FUNCTION_BLOCK FB_2001_doublecookie
VAR_INPUT
	execute: BOOL;
END_VAR
VAR
	TIMERDONE: BOOL;
END_VAR

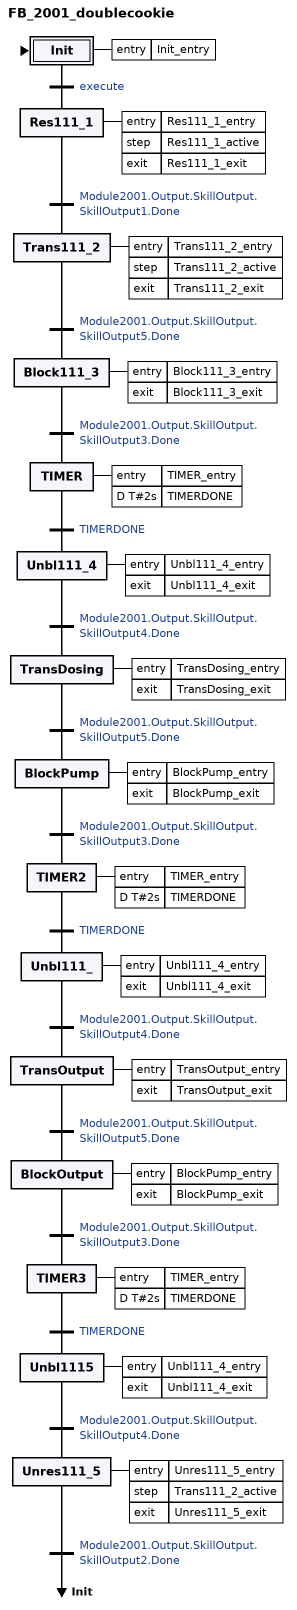
INITIAL_STEP Init:
    Init_entry(P1);  // entry action
END_STEP
TRANSITION FROM Init TO Res111_1
    := execute;
END_TRANSITION
STEP Res111_1:
    Res111_1_entry(P1);  // entry action
    Res111_1_active(N);  // step action
    Res111_1_exit(P0);  // exit action
END_STEP
TRANSITION FROM Res111_1 TO Trans111_2
    := Module2001.Output.SkillOutput.SkillOutput1.Done;
END_TRANSITION
STEP Trans111_2:
    Trans111_2_entry(P1);  // entry action
    Trans111_2_active(N);  // step action
    Trans111_2_exit(P0);  // exit action
END_STEP
TRANSITION FROM Trans111_2 TO Block111_3
    := Module2001.Output.SkillOutput.SkillOutput5.Done;
END_TRANSITION
STEP Block111_3:
    Block111_3_entry(P1);  // entry action
    Block111_3_exit(P0);  // exit action
END_STEP
TRANSITION FROM Block111_3 TO TIMER
    := Module2001.Output.SkillOutput.SkillOutput3.Done;
END_TRANSITION
STEP TIMER:
    TIMER_entry(P1);  // entry action
    TIMERDONE(D, T#2s);
END_STEP
TRANSITION FROM TIMER TO Unbl111_4
    := TIMERDONE;
END_TRANSITION
STEP Unbl111_4:
    Unbl111_4_entry(P1);  // entry action
    Unbl111_4_exit(P0);  // exit action
END_STEP
TRANSITION FROM Unbl111_4 TO TransDosing
    := Module2001.Output.SkillOutput.SkillOutput4.Done;
END_TRANSITION
STEP TransDosing:
    TransDosing_entry(P1);  // entry action
    TransDosing_exit(P0);  // exit action
END_STEP
TRANSITION FROM TransDosing TO BlockPump
    := Module2001.Output.SkillOutput.SkillOutput5.Done;
END_TRANSITION
STEP BlockPump:
    BlockPump_entry(P1);  // entry action
    BlockPump_exit(P0);  // exit action
END_STEP
TRANSITION FROM BlockPump TO TIMER2
    := Module2001.Output.SkillOutput.SkillOutput3.Done;
END_TRANSITION
STEP TIMER2:
    TIMER_entry(P1);  // entry action
    TIMERDONE(D, T#2s);
END_STEP
TRANSITION FROM TIMER2 TO Unbl111_
    := TIMERDONE;
END_TRANSITION
STEP Unbl111_:
    Unbl111_4_entry(P1);  // entry action
    Unbl111_4_exit(P0);  // exit action
END_STEP
TRANSITION FROM Unbl111_ TO TransOutput
    := Module2001.Output.SkillOutput.SkillOutput4.Done;
END_TRANSITION
STEP TransOutput:
    TransOutput_entry(P1);  // entry action
    TransOutput_exit(P0);  // exit action
END_STEP
TRANSITION FROM TransOutput TO BlockOutput
    := Module2001.Output.SkillOutput.SkillOutput5.Done;
END_TRANSITION
STEP BlockOutput:
    BlockPump_entry(P1);  // entry action
    BlockPump_exit(P0);  // exit action
END_STEP
TRANSITION FROM BlockOutput TO TIMER3
    := Module2001.Output.SkillOutput.SkillOutput3.Done;
END_TRANSITION
STEP TIMER3:
    TIMER_entry(P1);  // entry action
    TIMERDONE(D, T#2s);
END_STEP
TRANSITION FROM TIMER3 TO Unbl1115
    := TIMERDONE;
END_TRANSITION
STEP Unbl1115:
    Unbl111_4_entry(P1);  // entry action
    Unbl111_4_exit(P0);  // exit action
END_STEP
TRANSITION FROM Unbl1115 TO Unres111_5
    := Module2001.Output.SkillOutput.SkillOutput4.Done;
END_TRANSITION
STEP Unres111_5:
    Unres111_5_entry(P1);  // entry action
    Trans111_2_active(N);  // step action
    Unres111_5_exit(P0);  // exit action
END_STEP
TRANSITION FROM Unres111_5 TO Init
    := Module2001.Output.SkillOutput.SkillOutput2.Done;
END_TRANSITION

ACTION Block111_3_exit:
//BLOCKIEREN

Module2001.Input.SkillInput.SkillInput3.Execute := FALSE;
Module2001.Input.SkillInput.SkillInput3.ParameterInput.Parameterinput1.Value := 0; //TaskID
END_ACTION

ACTION TransDosing_entry:
//TRANSPORTIEREN

Module2001.Input.SkillInput.SkillInput5.Execute := TRUE;
Module2001.Input.SkillInput.SkillInput5.ParameterInput.Parameterinput1.Value := 3000; //X-Position
Module2001.Input.SkillInput.SkillInput5.ParameterInput.Parameterinput2.Value := 100;//90; //Z-Position
Module2001.Input.SkillInput.SkillInput5.ParameterInput.Parameterinput3.Value := 300; //Velocity
Module2001.Input.SkillInput.SkillInput5.ParameterInput.Parameterinput4.Value := 0; //Acceleration
END_ACTION

ACTION TransOutput_entry:
//TRANSPORTIEREN

Module2001.Input.SkillInput.SkillInput5.Execute := TRUE;
Module2001.Input.SkillInput.SkillInput5.ParameterInput.Parameterinput1.Value := 3300; //X-Position
Module2001.Input.SkillInput.SkillInput5.ParameterInput.Parameterinput2.Value := 110;//90; //Z-Position
Module2001.Input.SkillInput.SkillInput5.ParameterInput.Parameterinput3.Value := 300; //Velocity
Module2001.Input.SkillInput.SkillInput5.ParameterInput.Parameterinput4.Value := 0; //Acceleration
END_ACTION

ACTION TransOutput_exit:

Module2001.Input.SkillInput.SkillInput5.Execute := FALSE;
Module2001.Input.SkillInput.SkillInput5.ParameterInput.Parameterinput1.Value := 0; //X-Position
Module2001.Input.SkillInput.SkillInput5.ParameterInput.Parameterinput2.Value := 0; //Z-Position
Module2001.Input.SkillInput.SkillInput5.ParameterInput.Parameterinput3.Value := 0; //Velocity
Module2001.Input.SkillInput.SkillInput5.ParameterInput.Parameterinput4.Value := 0; //Acceleration
END_ACTION

ACTION Res111_1_entry:
// Reservieren entry
Module2001.Input.SkillInput.SkillInput1.Execute := TRUE;
Module2001.Input.SkillInput.SkillInput1.ParameterInput.Parameterinput1.Value := 111; //TASKID
END_ACTION

ACTION Block111_3_entry:
//BLOCKIEREN

Module2001.Input.SkillInput.SkillInput3.Execute := TRUE;
Module2001.Input.SkillInput.SkillInput3.ParameterInput.Parameterinput1.Value := 111; //TaskID
END_ACTION

ACTION Trans111_2_exit:
//TRANSPORTIEREN

Module2001.Input.SkillInput.SkillInput5.Execute := FALSE;
Module2001.Input.SkillInput.SkillInput5.ParameterInput.Parameterinput1.Value := 0; //X-Position
Module2001.Input.SkillInput.SkillInput5.ParameterInput.Parameterinput2.Value := 0; //Z-Position
Module2001.Input.SkillInput.SkillInput5.ParameterInput.Parameterinput3.Value := 0; //Velocity
Module2001.Input.SkillInput.SkillInput5.ParameterInput.Parameterinput4.Value := 0; //Acceleration
END_ACTION

ACTION Unbl111_4_exit:
//unBLOCKIEREN

Module2001.Input.SkillInput.SkillInput4.Execute := FALSE; 
Module2001.Input.SkillInput.SkillInput4.ParameterInput.Parameterinput1.Value := 000; //TaskID
END_ACTION

ACTION Unres111_5_entry:
//unreserve
Module2001.Input.SkillInput.SkillInput2.Execute := TRUE;
Module2001.Input.SkillInput.SkillInput2.ParameterInput.Parameterinput1.Value := 111; //TaskID
END_ACTION

ACTION Trans111_2_active:

END_ACTION

ACTION Init_entry:
execute := FALSE;
END_ACTION

ACTION BlockPump_entry:
//BLOCKIEREN

Module2001.Input.SkillInput.SkillInput3.Execute := TRUE;
Module2001.Input.SkillInput.SkillInput3.ParameterInput.Parameterinput1.Value := 111; //TaskID
END_ACTION

ACTION BlockPump_exit:
//BLOCKIEREN

Module2001.Input.SkillInput.SkillInput3.Execute := FALSE;
Module2001.Input.SkillInput.SkillInput3.ParameterInput.Parameterinput1.Value := 0; //TaskID
END_ACTION

ACTION Unres111_5_exit:
//unreserve
Module2001.Input.SkillInput.SkillInput2.Execute := FALSE;
Module2001.Input.SkillInput.SkillInput2.ParameterInput.Parameterinput1.Value := 0; //TaskID
END_ACTION

ACTION Trans111_2_entry:
//TRANSPORTIEREN

Module2001.Input.SkillInput.SkillInput5.Execute := TRUE;
Module2001.Input.SkillInput.SkillInput5.ParameterInput.Parameterinput1.Value := 2500; //X-Position
Module2001.Input.SkillInput.SkillInput5.ParameterInput.Parameterinput2.Value := 100;//90; //Z-Position
Module2001.Input.SkillInput.SkillInput5.ParameterInput.Parameterinput3.Value := 300; //Velocity
Module2001.Input.SkillInput.SkillInput5.ParameterInput.Parameterinput4.Value := 0; //Acceleration
END_ACTION

ACTION Res111_1_exit:
// Reservieren entry
Module2001.Input.SkillInput.SkillInput1.Execute := FALSE;
Module2001.Input.SkillInput.SkillInput1.ParameterInput.Parameterinput1.Value := 0; //TASKID
END_ACTION

ACTION TransDosing_exit:
//TRANSPORTIEREN

Module2001.Input.SkillInput.SkillInput5.Execute := FALSE;
Module2001.Input.SkillInput.SkillInput5.ParameterInput.Parameterinput1.Value := 0; //X-Position
Module2001.Input.SkillInput.SkillInput5.ParameterInput.Parameterinput2.Value := 0; //Z-Position
Module2001.Input.SkillInput.SkillInput5.ParameterInput.Parameterinput3.Value := 0; //Velocity
Module2001.Input.SkillInput.SkillInput5.ParameterInput.Parameterinput4.Value := 0; //Acceleration
END_ACTION

ACTION Res111_1_active:

END_ACTION

ACTION Unbl111_4_entry:
//unBLOCKIEREN

Module2001.Input.SkillInput.SkillInput4.Execute := TRUE; //FALSE weil timer
Module2001.Input.SkillInput.SkillInput4.ParameterInput.Parameterinput1.Value := 111; //TaskID
END_ACTION

ACTION TIMER_entry:
TIMERDONE := FALSE;
END_ACTION

END_FUNCTION_BLOCK

(* stored: Version 1.1.0.1, ProductVersion 3.1.0.25
   POU FB_2001_doublecookie: Id {8da49e05-89ab-4cc8-97ab-92307c4d85d5}
   Action Block111_3_exit: Id {1cf866cb-bd76-4bdf-b95a-a596e0acec35}
   Action TransDosing_entry: Id {428cd116-171d-4c64-8fe2-80763f4c8f4c}
   Action TransOutput_entry: Id {43285321-a067-495a-9571-923cb4cf216b}
   Action TransOutput_exit: Id {460096e8-1ead-49a9-ab79-2c4ac2001aa1}
   Action Res111_1_entry: Id {46818fb7-8f17-428f-ab65-56db59650ffd}
   Action Block111_3_entry: Id {4deb5a9b-15cc-41aa-bf4a-bacedef7484e}
   Action Trans111_2_exit: Id {4eaa4c2c-b8b1-41c8-80bb-2b22015c6f46}
   Action Unbl111_4_exit: Id {534c881c-19fd-43fe-90be-b609052cfe5a}
   Action Unres111_5_entry: Id {6bdfe5ab-f1fe-4eb3-a861-409cfecb5eda}
   Action Trans111_2_active: Id {75ea375c-e110-41ef-8052-40ad478454da}
   Action Init_entry: Id {8b407c86-d677-46a0-a90c-0c261a997188}
   Action BlockPump_entry: Id {8fe9ed49-6d78-4db7-af32-eb57d1402bbc}
   Action BlockPump_exit: Id {923cc8e1-fe70-4acb-801e-595f5286f4c3}
   Action Unres111_5_exit: Id {973b615b-c864-46f3-bee7-fc8465af5216}
   Action Trans111_2_entry: Id {a1d484c0-c565-4b20-85a6-5fa7e4bd8864}
   Action Res111_1_exit: Id {b652c482-3da9-4b9b-8edd-5d2d7f6f79d7}
   Action TransDosing_exit: Id {c33c45ef-e1ef-4db3-9996-0a789a8d4326}
   Action Res111_1_active: Id {d2b88d46-68fb-4df6-be3c-84f6c6d1aa64}
   Action Unbl111_4_entry: Id {e30795a1-9ad2-4f5b-bacc-03e854b367a2}
   Action TIMER_entry: Id {fb74a62b-134f-49b0-a769-2582a7fac839} *)
